FUNCTION_BLOCK TemperatureSensor
VAR
	stInputData			: MDP5001_320_A369A904;
	fOffsetInCelsius	: REAL;
END_VAR

{attribute 'monitoring' := 'call'}
PROPERTY Error : BOOL
GET
Error := stInputData.MDP5001_320_Input.MDP5001_320_Status.Error;
END_GET
END_PROPERTY

{attribute 'monitoring' := 'call'}
PROPERTY InCelsius : REAL
GET
InCelsius := (stInputData.MDP5001_320_Input.MDP5001_320_Value / 10.0) + fOffsetInCelsius;
END_GET
END_PROPERTY

{attribute 'monitoring' := 'call'}
PROPERTY InFarenheit : REAL
GET
InFarenheit := C_TO_F ( fX := InCelsius );
END_GET
END_PROPERTY

{attribute 'monitoring' := 'call'}
PROPERTY InKelvin : REAL
GET
InKelvin := C_TO_K ( fX := InCelsius );
END_GET
END_PROPERTY

{attribute 'monitoring' := 'call'}
PROPERTY InReaumur : REAL
GET
InReaumur := C_TO_R ( fX := InCelsius );
END_GET
END_PROPERTY

{attribute 'monitoring' := 'call'}
PROPERTY OffsetInCelsius : REAL
GET
OffsetInCelsius := fOffsetInCelsius;
END_GET
SET
fOffsetInCelsius := OffsetInCelsius;
END_SET
END_PROPERTY

{attribute 'monitoring' := 'call'}
PROPERTY Overrange : BOOL
GET
Overrange := stInputData.MDP5001_320_Input.MDP5001_320_Status.Overrange;
END_GET
END_PROPERTY

{attribute 'monitoring' := 'call'}
PROPERTY Underrange : BOOL
GET
Underrange := stInputData.MDP5001_320_Input.MDP5001_320_Status.Underrange;
END_GET
END_PROPERTY

END_FUNCTION_BLOCK

(* stored: Version 1.1.0.1
   POU TemperatureSensor: Id {0ed992bf-550f-455f-a941-ca8ef2257ea3}, SpecialFunc None
   Folder Status: Id {ce03e97b-142a-4b7a-a675-b138609ba55d}
   Folder Temperature: Id {08507647-4559-4ed5-86ad-63b7a9ffcad6}
   Property Error: Id {f1dcd065-a0e2-4942-b6be-52acd0d4f255}
   Get Get: Id {b7b1eee0-16eb-494f-b04a-3882a60ac41c}
   Property InCelsius: Id {36223012-ff55-4626-a711-0c8aed7cfcd9}
   Get Get: Id {ce133ee0-e068-4933-9973-245aa1226702}
   Property InFarenheit: Id {edb74bdf-3d63-4abe-9041-430a1c05d349}
   Get Get: Id {4d177a04-b64d-4ebf-87f5-90b61682804a}
   Property InKelvin: Id {a1d1c50b-431b-48e5-94b1-e93378b24ba4}
   Get Get: Id {85ef13f4-d165-4d4a-8f5c-538bda0361d2}
   Property InReaumur: Id {f5fc9271-aac9-4df7-ac7a-4e16f483dd53}
   Get Get: Id {d0171278-f08a-40bf-b826-6ec8f1f62072}
   Property OffsetInCelsius: Id {a94aef9d-f647-407e-b6d4-cc80386fd3ed}
   Get Get: Id {a3ae99d4-0c57-41b3-9f21-509ac98e195f}
   Set Set: Id {e257288e-b46d-4f62-a857-ed0f3d739963}
   Property Overrange: Id {61aade6e-6829-42c2-9b98-5ce3b9f9c02e}
   Get Get: Id {64bfaf44-59a1-46f8-b19e-8d346a414e5b}
   Property Underrange: Id {12278dfe-a928-4be5-947c-6989386e3bbf}
   Get Get: Id {3b14906d-682c-427a-9543-4b7b857b64e7} *)
